{attribute 'linkalways'} 
{attribute 'no_explicit_call' := 'This FB is a CLASS and must be accessed using methods or properties'}
{attribute 'enable_dynamic_creation'}
FUNCTION_BLOCK GetDatatypesRpcHandler IMPLEMENTS I_RpcHandler
VAR
	datatypes : I_Datatypes;
END_VAR

METHOD Handle
VAR_INPUT
	Parameters : I_Deserializer;
	Response : I_SynchronousRpcResponse;
END_VAR
VAR
	serializer : I_Serializer;
END_VAR
IF datatypes = 0 THEN
	Response.RejectWithMessage('GetDatatypesRpcHandler has not been initialized with a valid datatypes object');
	RETURN;
END_IF

serializer := Response.GetSerializer();
datatypes.SerializeTypeWith(serializer);
Response.CompleteWithSerializer(serializer);
serializer.Dispose();
END_METHOD

METHOD PUBLIC Initialize
VAR_INPUT
	Datatypes : I_Datatypes;
END_VAR
this^.datatypes := Datatypes;
END_METHOD

END_FUNCTION_BLOCK

(* stored: Version 1.1.0.1, ProductVersion 3.1.4024.12
   POU GetDatatypesRpcHandler: Id {fe657261-5aa9-4eea-b7e8-f9c0fc5dc57a}, SpecialFunc None
   Method Handle: Id {ac08dd12-42dd-424c-8b99-6d218ec38f4b}
   Method Initialize: Id {a7a5e8c5-5ad1-495d-854f-706ce0abdaac} *)
